PROGRAM MAIN
VAR

	SysRun					: BYTE;
	
END_VAR

SysRun := SysRun + 1;

EventLoggerManager();

RETURN;

END_PROGRAM

(* stored: Version 1.1.0.1, ProductVersion 3.1.4024.12
   POU MAIN: Id {0950bf5e-e2f0-4469-b3ab-cc3e91081a00}, SpecialFunc None *)
